Staubli VAL3: OnEvent16.pgx

program OnEvent16()
begin
  //-----------------------------------------------------------------------
  //Header begin
  //LasMAN3.7
  //Description of program
  //
  //Input parameters
  //
  //Output paramaters
  //Example
  //  call OnEvent1()
  //History
  //  Creation : 2013-06-23  y.ye@staubli.com
  //Header end
  //-----------------------------------------------------------------------
  resetMotion()
  if TxtFile:b8Axis
    // call Teach:Teach8Axis(TxtFile:trAxisData.rx,TxtFile:trAxisData.ry,0)
    call Teach:TeachAxis(TxtFile:trAxis8Data.x,TxtFile:trAxis8Data.y,TxtFile:trAxis8Data.z,TxtFile:trAxis8Data.rx,true)
  else
    popUpMsg("请到选项界面中激活八轴")
  endIf
  DataBase:nInterfaceType=9
end
